// TIA Portal V19 export
DATA_BLOCK "_IOL_1Par_rd_wrDI"   // DB116
AUTHOR : fur
FAMILY : IOL
VERSION : 0.0
// stored: AutoNumber false, InstanceOfName _IOL_1Par_rd_wr, InstanceOfType FB
"_IOL_1Par_rd_wr"
   // VAR_INPUT
   //    IA_Interface : Any;
   //    IHW_hwID : HW_ANY;
   //    II_CAP : Int;
   //    II_PORT : Int;
   //    I_DataStorage : Bool;
   //    I_BlockParam : Bool;
   //    IOL_INDEX : Int;
   //    IOL_SUBINDEX : Int;
   //    LEN : Int;
   // END_VAR
   // VAR_OUTPUT
   //    O_ComActiv : Bool;
   //    O_Fault : Bool;
   // END_VAR
   // VAR_IN_OUT
   //    IO_ReadReq : Bool;
   //    IO_WriteReq : Bool;
   //    IO_ResetReg : Bool;
   // END_VAR
   // VAR
   //    LIOLink_Call : "LIOLink_Device";
   //    DelCOMAct : TOF_TIME;
   //    SST_RecordData : Array[0..231] of Byte;
   //    STAT1 : Bool;
   //    Offset : DWord;
   //    S_NumberParameter : Int;
   //    S_NumberParameterSeq : Int;
   //    SI_StepAct : Int;
   //    SI_StepActSave : Int;
   //    SI_IOL_Index : Int;
   //    SI_IOL_Subindex : Int;
   //    SI_Len : Int;
   //    S_WordT : Word;
   //    S_StartParamDownload : Int;
   //    S_StartDeviceIdent : Int;
   //    S_StartAppSpezTag : Int;
   //    S_StartDeviceParam : Int;
   //    S_StartCommando : Int;
   //    S_NumberCommandos : Int;
   //    S_NumberComAct : Int;
   //    S_ByteT : Byte;
   //    IOL_Call_Busy : Bool;
   //    IOL_Call_Done_Valid : Bool;
   //    IOL_Call_Error : Bool;
   //    S_SeqActive : Bool;
   //    S_WriteActive : Bool;
   //    S_ReadActive : Bool;
   //    S_ComSeq : Bool;
   //    S_NoCom : Bool;
   //    S_FP_1 : Bool;
   //    S_RelRead : Bool;
   //    S_RelWrite : Bool;
   //    S_StartWrite : Bool;
   //    S_ReqDataStorBreak : Bool;
   //    S_ReqWriteCom : Bool;
   // END_VAR
BEGIN
END_DATA_BLOCK
